{attribute 'qualified_only'}
{attribute 'strict'}
{attribute 'to_string'}
TYPE MetricKind : (
	Gauge := 0,
	Counter := 1,
	UpDownCounter := 2
) UDINT;
END_TYPE

(* stored: Version 1.1.0.1
   DUT MetricKind: Id {a014bea1-bb58-4243-84bd-77ee1315ae72} *)
